Fanuc KAREL source: kt00928.KL

-- PROVISIONAL review KL for V1013-1; original PC SHA256 b57889dca82e4f3c466e456d9e48ef58e035bf844c1d2030c48275ade38a36fb
-- Incomplete behavior may be omitted. Consult companion uncertainty JSON. Do not deploy.
PROGRAM KT00928
%NOLOCKGROUP
VAR
  S1 : STRING[80]
  S2 : STRING[80]
  OUT : INTEGER
BEGIN
  -- UNRESOLVED_PC offsets 5-14; opcodes 3F,75
  -- UNRESOLVED_PC offsets 19-28; opcodes 3F,75
  -- UNRESOLVED_PC offsets 33-42; opcodes 3F,75
  -- UNRESOLVED_PC offsets 47-56; opcodes 3F,75
  -- UNRESOLVED_PC offsets 61-80; opcodes 27,22,2A,27,9D,76,23
  -- UNRESOLVED_PC offsets 85-89; opcodes 7F
END KT00928
